(* IEC 61131-3 sources: MotionTestBenchMaster/Logical/00_AID/Libraries/System_Libraries/powerlnk, 3 files *)

(* ---- powerlnk.typ ---- *)
(********************************************************************
 * COPYRIGHT -- Bernecker + Rainer
 ********************************************************************
 * Library: powerlnk
 * File: powerlnk.typ
 * Author: B+R
 ********************************************************************
 * Data types of library powerlnk
 ********************************************************************)

TYPE
	PLACTION_GET_DP_INFO_typ : STRUCT           (*query PDO info of datapoint *)
		DeviceName	: UDINT ;					(*in: pointer to the name of the I/O module holding the data point, e.g. "SS1.IF2.ST3.SL7"*)
		ChannelName	: UDINT ;					(*in: pointer to the name of the data point, e.g. "AnalogInput01"*)
		DestNode    : USINT ;                   (*out: Node number of destination *)
		SrcNode     : USINT ;                   (*out: Node number of source *)
		MessageType : USINT ;                   (*out: Message Type on Powerlink (3 PReq, 4 PRes) *)
		MuxSlot     : USINT ;                   (*out: multiplex slot (0 continous station) *)
		OffsetAbs   : UINT ;                    (*out: Offset in net data of EPL frame counted in bits *)
		OffsetRel   : UINT ;                    (*out: Offset relative to station net data in bits *)
		Length      : UINT ;                    (*out: Length of data point counted in bits *)
		TypeId      : UINT ;                    (*out: Type ident of datapoint EPL V2 (matches CANopen Specification) *)
		NodeInSize  : UINT ;                    (*out: input net size of station (Pres) *)
		NodeOutSize : UINT ;                    (*out: output net size of station (normally Preq) *)
		Direction   : USINT ;                   (*out: 1 Input, 2 Output relative to local node *)
		Node        : USINT ;                   (*out: node of datapoint *)
		reserved    : UINT ;                    (*res: reserved word for alignment *)
		ImageIndex  : UDINT ;                   (*out: image index for inputs 0 for outputs *)
		ImageOffset : UDINT ;                   (*out: offset of datapoint in local image buffer (bytes) *)
	END_STRUCT;
	PLACTION_GET_PDO_INFO_typ : STRUCT          (*query PDO info by index / subindex *)
		DeviceName	: UDINT ;					(*in: pointer to the name of the I/O module holding the data point, e.g. "SS1.IF2.ST3.SL7"*)
		ODIndex	    : UINT ;					(*in: Index of object in Powerlink object dictionary *)
		ODSubindex	: USINT ;					(*in: Subindex of object in Powerlink object dictionay *)
		align       : USINT ;                   (*res: reseved for alignment *)
		DestNode    : USINT ;                   (*out: Node number of destination *)
		SrcNode     : USINT ;                   (*out: Node number of source *)
		MessageType : USINT ;                   (*out: Message Type on Powerlink (3 PReq, 4 PRes) *)
		MuxSlot     : USINT ;                   (*out: multiplex slot (0 continous station) *)
		OffsetAbs   : UINT ;                    (*out: Offset in net data of EPL frame counted in bits *)
		OffsetRel   : UINT ;                    (*out: Offset relative to station net data in bits *)
		Length      : UINT ;                    (*out: Length of data point counted in bits *)
		TypeId      : UINT ;                    (*out: Type ident of datapoint EPL V2 (matches CANopen Specification) *)
		NodeInSize  : UINT ;                    (*out: input net size of station (Pres) *)
		NodeOutSize : UINT ;                    (*out: output net size of station (normally Preq) *)
		Direction   : USINT ;                   (*out: 1 Input, 2 Output relative to local node *)
		Node        : USINT ;                   (*out: node of datapoint *)
		reserved    : UINT ;                    (*res: reserved word for alignment *)
		ImageIndex  : UDINT ;                   (*out: image index for inputs 0 for outputs *)
		ImageOffset : UDINT ;                   (*out: offset of datapoint in local image buffer (bytes) *)
	END_STRUCT;
	PLACTION_GET_CROSSLINK_INFO_typ : STRUCT	(*query position of I/O data points in the poll response frame to listen in on inputs from other CNs*)
		DeviceName	: UDINT ;					(*in: pointer to the name of the I/O module holding the data point, e.g. "SS1.IF2.ST3.SL7"*)
		ChannelName	: UDINT ;					(*in: pointer to the name of the data point, e.g. "AnalogInput01"*)
		NodeId	: UINT ;						(*out: node number of POWERLINK station*)
		Offset	: UINT ;						(*out: offset in the data range of the poll response frames in bits*)
		Length	: UINT ;						(*out: size of the data point in the poll response frame in bits*)
		TypeId	: UINT ;						(*out: data type ident of the data point according to the V2 specification*)
	END_STRUCT;
	PLACTION_DEVICE_TO_BUS_NR_typ : STRUCT		(*determines the POWERLINK bus number from the device definition*)
		pDeviceString	: UDINT ;				(*in: string with the device definition in the form "SLx.SSy.IFz", e.g. "SL0.SS1.IF1", given as a pointer, *)
		busNumber	: USINT ;					(*out: after the function is called, the POWERLINK bus number is in this structure element*)
	END_STRUCT;
	PLACTION_SYNC_STATISTICS_typ : STRUCT		(*reads the times of the synchronous task class*)
		act_usec	: UINT ;					(*out: execution period during the last measured cycle*)
		min_usec	: UINT ;					(*out: minimum execution period*)
		max_usec	: UINT ;					(*out: maximum execution period*)
		act_cycle	: UINT ;					(*out: cycle time during the last measured cycle*)
		min_cycle	: UINT ;					(*out: minimum cycle time*)
		max_cycle	: UINT ;					(*out: maximum cycle time*)
	END_STRUCT;
	PLSYSCONF_RS_typ : STRUCT					(*this structure is only evaluated on SG3 targets*)
		size_x16	: USINT ;					(*size of the configuration entry in 16 byte blocks*)
		bus	: USINT ;							(*bus number where the remote station is located*)
		station	: USINT ;						(*station number of the station*)
		flags	: USINT ;						(*parameter flags for the station: 16#00 normal station, 16#20 slow station*)
		hwVariant	: UDINT ;					(*hardware variant ID *)
		insize	: INT ;							(*input buffer size of the station*)
		outsize	: INT ;							(*output buffer size of the station*)
		RespTimeout	: INT ;						(*response timeout in µs*)
		MuxNetworkSlot	: USINT ;				(*ignored for normal stations, for multiplexed stations 1 to MuxPrescaler*)
		reserve2	: USINT ;					(*reserved for future updates*)
	END_STRUCT;
	PLACTION_GET_IDENT_typ : STRUCT				(*determines a station ID*)
		pName	: UDINT ;						(*string with the station description, e.g. "SL0.SS1.IF1", given as a pointer*)
		ident	: UDINT ;						(*after the function is called, the station ID is located in this structure element*)
	END_STRUCT;
	PLACTION_NET_QUALITY_typ : STRUCT			(*reads statistic information regarding network quality*)
		nLineQualFreezeCnt	: UDINT ;			(*number of POWERLINK cycles in during the measurement period*)
		nLineQualFailCnt	: UDINT ;			(*number of failed POWERLINK cycles*)
	END_STRUCT;
	PLSYSCONF_IF_typ : STRUCT					(*determines configured POWERLINK interface parameters*)
		station	: USINT ;						(*station number: 0 for manager, 1...253 for controllers*)
		slot	: USINT ;						(*slot of the POWERLINK interface card*)
		subslot	: USINT ;						(*subslot of the POWERLINK interface card*)
		interface	: USINT ;					(*interface number*)
		pl_cycle	: UDINT ;					(*cycle time of a POWERLINK network cycle*)
		pl_prescale	: UDINT ;					(*prescaler for synchronous task classes*)
		uptimeout	: UDINT ;					(*timeout defining how long the wait should be when booting the slave*)
		bus	: USINT ;							(*bus number for this interface*)
		MuxStationsPerCycle	: USINT ;			(*number of multiplexed stations per POWERLINK cycle*)
		MuxPrescaler	: USINT ;				(*number of POWERLINK cycles for one mux cycle 1 .. 253*)
		ATOCtaskclass	: SINT ;				(*taskclass triggering the Output-DMA, 0 ..triggered by System-Tick, plCE_CYCLIC_1 to plCE_CYCLIC_8 ..triggered by cyclic taskklass*)
		reservedlong	: UDINT ;				(*reserved*)
	END_STRUCT;
	PLSYSCONF_typ : STRUCT						(*configuration structure which must be transferred to plConfig*)
		noIF	: USINT ;						(*number of interface cards*)
		takt_master	: USINT ;					(*specifies which interface card should trigger the synchronous timer2 task class*)
		reserve1	: UINT ;					(*reserved for future use (should always be set to 0)*)
		pRemoteCfg	: UDINT ;					(*pointer to an array with remote station configurations*)
		interfaces	: ARRAY[0..14] OF PLSYSCONF_IF_typ ;	(*interface configurations*)
	END_STRUCT;
END_TYPE

(* ---- powerlnk.fun ---- *)
(********************************************************************
 * COPYRIGHT -- Bernecker + Rainer
 ********************************************************************
 * Library: powerlnk
 * File: powerlnk.fun
 * Author: B+R
 ********************************************************************
 * Functions and function blocks of library powerlnk
 ********************************************************************)

{REDUND_CONTEXT} {REDUND_UNREPLICABLE} FUNCTION plAction : UINT					(*triggers events and reads statistic information*)
	VAR_INPUT
		ident	:UDINT;						(*identifier for which the action should be triggered*)
		actionID	:UDINT;					(*ID number of the action which should be triggered*)
		pObject	:UDINT;						(*pointer to the structure in which the parameters and return values of the action are entered*)
		objectLen	:UDINT;					(*size of the structure which was specified with pObject*)
	END_VAR
END_FUNCTION
{REDUND_CONTEXT} {REDUND_UNREPLICABLE} FUNCTION plState : UINT						(*queries status*)
	VAR_INPUT
		ident	:UDINT;						(*identifier of a data point, identifier of a non-cyclic channel or POWERLINK station identifier*)
	END_VAR
END_FUNCTION
{REDUND_CONTEXT} {REDUND_UNREPLICABLE} FUNCTION plAcycWrite : UINT					(*submits data on a non-cyclic communication channel*)
	VAR_INPUT
		ident	:UDINT;						(*identifier returned from plAcycOpen*)
		bufferAdr	:UDINT;					(*pointer to the buffer which should be written*)
		bufferLen	:UDINT;					(*number of bytes which should be written*)
		pWrittenLen	:REFERENCE TO UDINT;	(*pointer to the number of actual written bytes*)
	END_VAR
END_FUNCTION
{REDUND_CONTEXT} {REDUND_UNREPLICABLE} FUNCTION plAcycInvite : UINT				(*requests data on a non-cyclic communication channel*)
	VAR_INPUT
		ident	:UDINT;						(*identifier returned from plAcycOpen*)
	END_VAR
END_FUNCTION
{REDUND_CONTEXT} {REDUND_UNREPLICABLE} FUNCTION plAcycRead : UINT					(*reads data on a non-cyclic communication channel*)
	VAR_INPUT
		ident	:UDINT;						(*identifier returned from plAcycOpen*)
		bufferAdr	:UDINT;					(*pointer to the buffer where reading should take place*)
		bufferLen	:UDINT;					(*maximum number of bytes which should be read*)
		pReadLen	:REFERENCE TO UDINT;	(*pointer to the number of actual read bytes*)
	END_VAR
END_FUNCTION
{REDUND_CONTEXT} {REDUND_UNREPLICABLE} FUNCTION plAcycClose : UINT					(*closes a non-cyclic communication channel*)
	VAR_INPUT
		ident	:UDINT;						(*identifier returned from plAcycOpen()*)
	END_VAR
END_FUNCTION
{REDUND_CONTEXT} {REDUND_UNREPLICABLE} FUNCTION plAcycOpen : UINT					(*opens a non-cyclic communication channel*)
	VAR_INPUT
		pName	:STRING[80];				(*pointer to the station and channel name which should be written to or read from*)
		flags	:UDINT;						(*e.g. plOPEN_MODE_READ = read, plOPEN_MODE_WRITE = write, ...*)
		pIdent	:REFERENCE TO UDINT;		(*pointer to the ID of the opened channel*)
	END_VAR
END_FUNCTION
{REDUND_CONTEXT} {REDUND_UNREPLICABLE} FUNCTION plCEDelete : UINT					(*deletes a cyclic copy instruction*)
	VAR_INPUT
		ident	:UDINT;						(*identifier returned from plCECreate*)
	END_VAR
END_FUNCTION
{REDUND_CONTEXT} {REDUND_UNREPLICABLE} FUNCTION plCECreate : UINT					(*creates a cyclic copy instruction*)
	VAR_INPUT
		pDatapoint	:STRING[80];			(*pointer to the string with a data point definition*)
		address	:UDINT;						(*pointer to the image from/to which the value of the IO data point should be copied*)
		taskclass	:SINT;					(*e.g. plCE_CYCLIC_1 = Cyclic #1, plCE_CYCLIC_2 = Cyclic #2, ...*)
		pIdent	:REFERENCE TO UDINT;		(*pointer to the ID where the created data point should be returned*)
	END_VAR
END_FUNCTION
{REDUND_CONTEXT} {REDUND_UNREPLICABLE} FUNCTION plConfig : UINT					(*sets the POWERLINK configuration*)
	VAR_INPUT
		pConfigStruct	:UDINT;				(*pointer to the configuration structure*)
	END_VAR
END_FUNCTION

(* ---- powerlnk.var ---- *)
(********************************************************************
 * COPYRIGHT -- Bernecker + Rainer
 ********************************************************************
 * Library: powerlnk
 * File: powerlnk.var
 * Author: B+R
 ********************************************************************
 * Local variables of library powerlnk
 ********************************************************************)

VAR CONSTANT
	ERR_PLMGR_VERS_CONFLICT         : UINT	:= 20900;		(*version conflict in the memory structure*)
	ERR_PLMGR_NOMEM                 : UINT	:= 20901;		(*error allocating memory*)
	ERR_PLMGR_WRONG_DEVICE          : UINT	:= 20903;		(*incorrect device definition*)
	ERR_PLMGR_CONFIG_NOT_FOUND      : UINT	:= 20904;		(*configuration was not found*)
	ERR_PLMGR_ALREADY_CONFIGURATED  : UINT	:= 20905;		(*configuration already carried out*)
	ERR_PLMGR_NOT_IMPLEMENTED       : UINT	:= 20906;		(*desired function is not supported*)
	ERR_PLMGR_ILLEGAL_PARAMETER     : UINT	:= 20908;		(*invalid parameter given to the function*)
	ERR_PLMGR_WRONG_IDENT           : UINT	:= 20911;		(*incorrect or invalid ident given*)
	ERR_PLMGR_ERROR_ALLOC_STATION   : UINT	:= 20913;		(*station allocation failed*)
	ERR_PLMGR_ERROR_ALLOC_CHANNEL   : UINT	:= 20914;		(*allocating the non-cyclic communication channel failed*)
	ERR_PLMGR_ERROR_ALLOC_BUFFER    : UINT	:= 20915;		(*allocating the buffer failed*)
	ERR_PLMGR_CHANNEL_ALREADY_OPEN  : UINT	:= 20916;		(*non-cyclic communication channel is already open*)
	ERR_PLMGR_NO_FRAME_RECEIVED     : UINT	:= 20917;		(*no frame ready to be called*)
	ERR_PLMGR_FRAME_TOO_LONG        : UINT	:= 20918;		(*the frame to be sent is larger than the buffer used to transfer it*)
	ERR_PLMGR_WRITE_ACTIVE          : UINT	:= 20919;		(*previous write on this channel was not completed*)
	ERR_PLMGR_OFFSET_TO_HIGH        : UINT	:= 20920;		(*offset too large for ident*)
	ERR_PLMGR_NIL_POINTER           : UINT	:= 20921;		(*NIL pointer given as a parameter*)
	ERR_PLMGR_OVERFLOW              : UINT	:= 20922;		(*buffer overflow*)
	ERR_PLMGR_UNAVAILABLE_DATAPOINT : UINT	:= 20923;		(*data point not available*)
	ERR_PLMGR_WRONG_TASKCLASS       : UINT	:= 20924;		(*incorrect task class*)
	ERR_PLMGR_STATION_NOT_ACTIVE    : UINT	:= 20925;		(*station not active*)
	ERR_PLMGR_TOO_MANY_INTERFACES   : UINT	:= 20926;		(*too many POWERLINK interfaces are configured*)
	ERR_PLMGR_BUS_CONFIGURED_TWICE  : UINT	:= 20927;		(*bus number configured twice*)
	ERR_PLMGR_SYNC_BY_SYSTEM        : UINT	:= 20928;		(*synchronization must take place using the system configuration*)
	ERR_PLMGR_SYNC_FAILED           : UINT	:= 20929;		(*synchronizing the task class system failed*)
	ERR_PLMGR_CONFIG_CONFLICT       : UINT	:= 20930;		(*IOTIMER device configuration failed (synchronization)*)
	ERR_PLMGR_NOT_IN_PRES           : UINT	:= 20931;		(*specified data point is not in the station's poll response frame and can therefore not be heard*)
	ERR_PLMGR_UNKNOWN_TYPE          : UINT	:= 20932;		(*datatype of data point not valid*)
	ERR_PLMGR_NO_PDO_MAPPING_DEFINED: UINT	:= 20933;		(*no PDO mapping defined*)
	ERR_PLMGR_PARSE_ERROR           : UINT	:= 20950;		(*error parsing the data point definition*)
	ERR_PLMGR_PARSE_END_EXPECTED    : UINT	:= 20951;		(*data point definition continues past an expected end*)
	ERR_PLMGR_PARSE_NO_PERCENT      : UINT	:= 20952;		(*no % at the beginning of the data point definition*)
	ERR_PLMGR_PARSE_NOT_IN_OR_OUT   : UINT	:= 20953;		(*direction specification in the data point definition is neither IN (I) nor OUT (Q)*)
	ERR_PLMGR_PARSE_INTERFACE       : UINT	:= 20954;		(*incorrect interface number*)
	ERR_PLMGR_PARSE_STATION         : UINT	:= 20955;		(*incorrect station number*)
	ERR_PLMGR_PARSE_MODUL           : UINT	:= 20956;		(*incorrect module number*)
	ERR_PLMGR_PARSE_SUBMODUL        : UINT	:= 20957;		(*invalid submodule or screw-in slot number*)
	ERR_PLMGR_PARSE_CHANNEL         : UINT	:= 20958;		(*incorrect channel number*)
	ERR_PLMGR_PARSE_BIT             : UINT	:= 20959;		(*incorrect bit number*)
	ERR_PLMGR_PARSE_TO_MANY_NUMBERS : UINT	:= 20960;		(*too many numbers in the data point definition*)
	ERR_PLMGR_PARSE_NETTIME         : UINT	:= 20961;		(*incorrect data type or length for NETTIME*)
	ERR_PLMGR_PARSE_SLOT            : UINT	:= 20962;		(*incorrect slot number*)
	ERR_PLMGR_PARSE_SUBSLOT         : UINT	:= 20963;		(*incorrect subslot number*)
	ERR_PLMGR_PARSE_TRAILINGCHARS   : UINT  := 20964;       (*characters follow a valid channel or device name*)
	ERR_PLMGR_PARSE_ARRAYSIZE       : UINT  := 20965;       (*arraysize not valid*)
	ERR_PLMGR_WARNING_FW_UPDATE     : UINT	:= 20980;		(*firmware update executed for the station (in error logbook)*)
	ERR_PLMGR_HW_BOOTUP_FAILED      : UINT	:= 20981;		(*error when starting POWERLINK hardware (in error logbook)*)
	ERR_PLMGR_RECOMMEND_FW_UPDATE   : UINT	:= 20982;		(*update for the IF686 recommended; download the current plfif686.br file*)
	ERR_PLMGR_INTERNAL              : UINT	:= 20997;		(*internal error which should never occur (in error logbook)*)
	ERR_PLMGR_EXCEPTION             : UINT	:= 20998;		(*exception from POWERLINK hardware (in error logbook)*)
	ERR_PLMGR_NO_POWERLNK_LIBRARY   : UINT	:= 20999;		(*powerLnk library not loaded at this time*)
	plACTION_GET_NET_QUALITY        : UDINT	:= 1;			(*reads the connection quality*)
	plACTION_GET_IDENT              : UDINT	:= 2;			(*determines a station ID*)
	plACTION_START_SYNC_STATISTICS  : UDINT	:= 3;			(*switches on time measurement for synchronous task classes*)
	plACTION_STOP_SYNC_STATISTICS   : UDINT	:= 4;			(*switches off time measurement for synchronous task classes*)
	plACTION_GET_SYNC_STATISTICS    : UDINT	:= 5;			(*reads time measurement values for synchronous task classes*)
	plACTION_GET_FIRMWARE_VERSION   : UDINT	:= 6;			(*reads the firmware version from the POWERLINK hardware*)
	plACTION_DEVICE_TO_BUS_NR       : UDINT	:= 7;			(*derives the bus number from the device definition 'SLx.SSy.IFz'*)
	plACTION_GET_STATION_NUMBER     : UDINT	:= 8;			(*reads the station number of the local station into a UDINT variable*)
	plACTION_GET_IF_PARAMETERS      : UDINT	:= 9;			(*reads interface parameters for a POWERLINK interface to a PLSYSCONF_IF_typ structure*)
	plACTION_GET_STATIONFLAG        : UDINT	:= 12;			(*checks flag for a POWERLINK station*)
	plACTION_GET_STATION_HWVARIANT  : UDINT	:= 13;			(*reads the POWERLINK station hardware variant*)
	plACTION_GET_IF_CYCLE_TIME      : UDINT	:= 15;			(*reads the set POWERLINK cycle time in µs*)
	plACTION_GET_IF_PRESCALE        : UDINT	:= 16;			(*reads the set POWERLINK prescaler*)
	plACTION_GET_IF_MUXPRESCALE     : UDINT	:= 17;			(*reads the multiplexed prescaler*)
	plACTION_GET_IF_RSQUEUELAPCNT   : UDINT	:= 18;			(*get rs queue lap count to UDINT variable*)
	plACTION_GET_CROSSLINK_INFO     : UDINT	:= 19;			(*query the cross-communication information of an I/O data point*)
	plACTION_GET_DP_INFO            : UDINT := 21;			(*query the PDO information of an I/O data point*)
	plACTION_GET_PDO_INFO           : UDINT := 22;			(*query the PDO information of by Index/Subindex*)

	plDIRECTION_IN                  : USINT := 1;			(*Direction "input" to PLC returned from plACTION_GET_PDO_INFO *)
	plDIRECTION_OUT                 : USINT := 2;     (*Direction "output" from PLC returned from plACTION_GET_PDO_INFO *)
	plDIRECTION_XOUT                : USINT := 3;     (*Direction "crosslinked output" returned from plACTION_GET_PDO_INFO *)
	plMESSAGE_TYPE_PREQ             : USINT	:= 3;	    (*MessageType "poll request" returned from plACTION_GET_PDO_INFO *)
	plMESSAGE_TYPE_PRES             : USINT	:= 4;     (*MessageType "poll response" returned from plACTION_GET_PDO_INFO *)

	plSTATE_CHANNEL_READ_MASK       : UINT	:= 16#00F0;		(*mask which conceals the read conditions on non-cyclic RW channels*)
	plSTATE_CHANNEL_READ_CLOSED     : UINT	:= 16#0000;		(*this non-cyclic channel is not open for read access*)
	plSTATE_CHANNEL_READ_EMPTY      : UINT	:= 16#0010;		(*there are no messages on this non-cyclic channel to be picked up*)
	plSTATE_CHANNEL_READ_READY      : UINT	:= 16#0020;		(*there are messages present to be picked up with plAcycRead() on this non-cyclic channel*)
	plSTATE_CHANNEL_READ_WRONG      : UINT	:= 16#00F0;		(*outcome from AND connector between plSTATE_WRONG_IDENT and plSTATE_CHANNEL_READ_MASK*)

	plSTATE_CHANNEL_WRITE_MASK      : UINT	:= 16#0f00;		(*mask which conceals the write conditions on non-cyclic RW channels*)
	plSTATE_CHANNEL_WRITE_CLOSED    : UINT	:= 16#0000;		(*this non-cyclic channel is not open for write access*)
	plSTATE_CHANNEL_WRITE_ACTIVE    : UINT	:= 16#0200;		(*current write access on this non-cyclic channel is being processed*)
	plSTATE_CHANNEL_WRITE_OPEN      : UINT	:= 16#0100;		(*this non-cyclic channel is opened for write access, but none have taken place so far*)
	plSTATE_CHANNEL_WRITE_WRONG     : UINT	:= 16#0f00;		(*outcome from AND connector between plSTATE_WRONG_IDENT and plSTATE_CHANNEL_WRITE_MASK*)

	plSTATE_STATION_NONEXISTANT     : UINT	:= 0;			(*station was not previously addressed*)
	plSTATE_STATION_WAITING         : UINT	:= 1;			(*station picked up by the software but not yet reported to the bus*)
	plSTATE_STATION_OSDL            : UINT	:= 2;			(*new firmware has just been loaded to the station*)
	plSTATE_STATION_CONFIG          : UINT	:= 3;			(*station is online but no cyclic instructions have been carried out so far*)
	plSTATE_STATION_ACTIVATEING     : UINT	:= 4;			(*the station has just been activated*)
	plSTATE_STATION_ACTIVE          : UINT	:= 5;			(*station is online and cyclic copy instructions are carried out*)
	plSTATE_STATION_INACTIVE        : UINT	:= 6;			(*station no longer online although it had just been ACTIVE*)
	plSTATE_STATION_CHANGED         : UINT	:= 7;			(*the hardware configuration for the station was changed*)
	plSTATE_STATION_CFGFAILED       : UINT	:= 8;			(*the configuration of the station failed, and the option EPL_NoResetOnConfigFail is on. *)
	plSTATE_STATION_FAILED          : UINT	:= 15;			(*station configuration failed with a fatal error*)

	plSTATE_CE_WAITING              : UINT	:= 1;			(*copy entry is activated as soon as a station becomes active*)
	plSTATE_CE_ACTIVE               : UINT	:= 2;			(*copy entry active*)
	plSTATE_CE_INACTIVE             : UINT	:= 3;			(*copy entry was active but the station was inactive in the meantime*)
	plSTATE_CE_ERROR                : UINT	:= 4;			(*copy entry faulty, e.g. offset too large or module not present on this station*)

	plSTATE_WRONG_IDENT             : UINT	:= 65535;		(*return value which an incorrect ID is transferred*)

	plSYSCONF_STATIONFLAG_SLOW      : USINT	:= 16#20;		(*station is a multiplexed station*)

	plOPEN_MODE_READ                : UDINT	:= 0;			(*'read' mode for plAcycOpen()*)
	plOPEN_MODE_WRITE               : UDINT	:= 1;			(*'write' mode for plAcycOpen()*)
	plOPEN_MODE_RW                  : UDINT	:= 2;			(*'read/write' mode for plAcycOpen()*)
	plOPEN_MODE_EPLV1               : UDINT	:= 16;			(*no effect for V1 networks*)
	plOPEN_MODE_EPLV2               : UDINT	:= 32;			(*allows aSend frames to be sent and received on this channel*)
	plOPEN_MODE_LENGTH              : UDINT	:= 64;			(*causes the length of the net data to be entered on the first 2 bytes for V2 frames as well*)

	plCE_TIMER_1                    : SINT	:= -1;			(*task class timer#2 for plCECreate()*)
	plCE_TIMER_2                    : SINT	:= -2;			(*task class timer#1 for plCECreate()*)
	plCE_CYCLIC_1                   : SINT	:= 1;			(*task class cyclic#1 for plCECreate()*)
	plCE_CYCLIC_2                   : SINT	:= 2;			(*task class cyclic#2 for plCECreate()*)
	plCE_CYCLIC_3                   : SINT	:= 3;			(*task class cyclic#3 for plCECreate()*)
	plCE_CYCLIC_4                   : SINT	:= 4;			(*task class cyclic#4 for plCECreate()*)
	plCE_CYCLIC_5                   : SINT	:= 5;			(*task class cyclic#5 for plCECreate()*)
	plCE_CYCLIC_6                   : SINT	:= 6;			(*task class cyclic#6 for plCECreate()*)
	plCE_CYCLIC_7                   : SINT	:= 7;			(*task class cyclic#7 for plCECreate()*)
	plCE_CYCLIC_8                   : SINT	:= 8;			(*task class cyclic#8 for plCECreate()*)
END_VAR
